FUNCTION_BLOCK FB_Observable_REAL EXTENDS FB_AbstractObservable
VAR
    _fVal:                  REAL;
END_VAR

PROPERTY fValue32 : REAL
GET
fValue32 := THIS^._fVal;
END_GET
SET
THIS^._fVal := fValue32;

IF THIS^._bAutoNotify THEN
    THIS^.Notify();
END_IF
END_SET
END_PROPERTY

METHOD  Notify : I_Observable
VAR
    i:      UDINT;
END_VAR
Notify := THIS^;

IF THIS^.nObserverCount <= 0 THEN
    RETURN;
END_IF

FOR i := 0 TO THIS^.nLastIdx DO
    THIS^.pipObserver[i].Update(THIS^._fVal);
END_FOR
END_METHOD

METHOD  NotifyLast : I_Observable
NotifyLast := THIS^;

IF THIS^.nObserverCount <= 0 THEN
    RETURN;
END_IF

THIS^.pipObserver[THIS^.nLastIdx].Update(THIS^._fVal);
END_METHOD

END_FUNCTION_BLOCK

(* stored: Version 1.1.0.1, ProductVersion 3.1.4024.12
   POU FB_Observable_REAL: Id {44f2149a-e556-4278-8e29-b5be8430ad03}, SpecialFunc None
   Property fValue32: Id {a0813b3d-f5d1-4dc2-abb7-e188f52cb384}
   Get Get: Id {1b7554b4-9021-4d07-9c73-8d38b15ac4db}
   Set Set: Id {2a2e589f-9528-41d6-9e71-704813bd50f0}
   Method Notify: Id {bdb8eebc-0456-495a-bfc0-8db8495e80d3}
   Method NotifyLast: Id {d836ad80-4747-45ab-acac-519a63f75d6b} *)
